FUNCTION_BLOCK FB_Btn
VAR_INPUT
 (*exemple : Btn                                                             :FB_BtnHmiType; (**)*)

	HmiStart:			FB_BtnHmiAutoResetType; (*Start button*)
	HmiStop:			FB_BtnHmiAutoResetType; (*Stop button*)
	HmiReset:			FB_BtnHmiAutoResetType;
	ResetAllHoming:		FB_BtnHmiAutoResetType;
	Init:				FB_BtnHmiAutoResetType; (*Start button*)
	Man:				FB_BtnHmiAutoResetType; (*Stop button*)
	Auto:				FB_BtnHmiAutoResetType; (*Reset button*)
//	Step:				FB_BtnHmiAutoResetType; (*Set step by step mode*)




(************************************************************************************)
(*      Boutons du mode manuel                                                                                *)
(************************************************************************************)

END_VAR
VAR_OUTPUT
END_VAR
VAR

END_VAR

HmiStart();
HmiStop();(**)
HmiReset();(**)
ResetAllHoming();
Init();
Auto();
Man();
//Step(); (**)

END_FUNCTION_BLOCK

(* stored: Version 1.1.0.1, ProductVersion 3.1.4020.12
   POU FB_Btn: Id {219ce889-16ba-497c-b7d0-df2e74ec6ee2}, SpecialFunc None *)
